{attribute 'linkalways'} 
{attribute 'no_explicit_call' := 'This FB is a CLASS and must be accessed using methods or properties'}
{attribute 'enable_dynamic_creation'}
FUNCTION_BLOCK INTERNAL MoveAdditiveCommand EXTENDS MoveCommand
VAR
	_fb : MC_MoveAdditive;
	_distance : LREAL;
END_VAR

METHOD FB_init : BOOL
VAR_INPUT
	bInitRetains : BOOL; // if TRUE, the retain variables are initialized (warm start / cold start)
	bInCopyCode : BOOL;  // if TRUE, the instance afterwards gets moved into the copy code (online change)
	axis : I_Axis;
	distance : LREAL;
	velocity : LREAL;
	acceleration : LREAL;
	deceleration : LREAL;
	jerk : LREAL;
	bufferMode : AxisBufferMode;
END_VAR
_axis := axis;
_distance := distance;
_velocity := velocity;
_acceleration := acceleration;
_deceleration := deceleration;
_jerk := jerk;
_bufferMode := bufferMode;
END_METHOD

PROPERTY PUBLIC IsActive : BOOL
GET // PUBLIC
IsActive := _fb.Active;
END_GET
END_PROPERTY

METHOD PROTECTED OnExecuting
VAR_INPUT
	stateControl : I_AsyncCommandStateControl;
END_VAR
_fb(
	Axis := _axis._InternalAxisRef,
	Execute := TRUE,
	Distance := _distance,
	Velocity := _velocity,
	Acceleration := _acceleration,
	Deceleration := _deceleration,
	Jerk := _jerk,
	BufferMode := _bufferMode
);

IF _fb.Busy THEN
	RETURN;
END_IF

_fb(Axis := _axis._InternalAxisRef, Execute := FALSE);

IF _fb.CommandAborted THEN
	THIS^.Abort();
	RETURN;
END_IF

IF _fb.Error THEN
	stateControl.Error(_fb.ErrorID);
	RETURN;
END_IF

stateControl.Next();
END_METHOD

END_FUNCTION_BLOCK

(* stored: Version 1.1.0.1, ProductVersion 3.1.4024.12
   POU MoveAdditiveCommand: Id {d419e8ad-959a-4135-8dc0-59c8c9a95e25}, SpecialFunc None
   Folder Constructor: Id {a73fdce8-d501-4bec-bbd1-8c2171dc8711}
   Method FB_init: Id {f129428b-69fb-4083-bf50-df32f60c42f4}
   Property IsActive: Id {c9e83266-0349-0304-0873-2616d32bceb4}
   Get Get: Id {1ed032a1-391b-0c16-086d-aeded9550c3e}
   Method OnExecuting: Id {8f46bf76-d026-0863-2a89-ed39fff444c3} *)
